// TIA Portal V18 export
TYPE "UDT_MES_Monitoring_station"
   STRUCT
      StationName : String := 'Station X';
      CheckIn : Struct
         Req : Bool;
         OK : Bool;
         NG : Bool;
         Done : Bool;
         InProgress : Bool;
         Timeout : Bool;
         Elapsed : Time;
         BothOkNg : Bool;
         UnexpectedDone : Bool;
         CountOK : UDInt;
         CountNG : UDInt;
         CountDone : UDInt;
         CountTimeout : UDInt;
         DATA : Struct
            PLC_PartTypeID : Int;
            PLC_StationRecipeNo : Int;
            PLC_StationDMXCode : String[128];
            PLC_StationStatus : Int;
            MES_ErrorCode : Int;
            MES_StatusBits : DInt;
            MES_Cycle_ID : DInt;
            MES_Unit_ParttypeID : Int;
         END_STRUCT;
      END_STRUCT;
      CheckOut : Struct
         Req : Bool;
         StoredOK : Bool;
         StoredNG : Bool;
         Done : Bool;
         InProgress : Bool;
         Timeout : Bool;
         Elapsed : Time;
         BothOkNg : Bool;
         UnexpectedDone : Bool;
         CountOK : UDInt;
         CountNG : UDInt;
         CountDone : UDInt;
         CountTimeout : UDInt;
         DATA : Struct
            PLC_PartTypeID : Int;
            PLC_StationDMXCode : String[50];
            PLC_StationRecipeNo : Int;
            PLC_PartStatus : Int;
            PLC_SubPartSN1 : String[50];
            PLC_TransferTime : String[50];
            PLC_Power : Real;
            PLC_Displacement : Real;
            PLC_Program : Int;
            PLC_NGCode : Int;
            MES_ErrorCode : Int;
            MES_ErrorMsg : String[60];
         END_STRUCT;
      END_STRUCT;
      SubPart : Struct
         OK : Bool;
         NG : Bool;
         Done : Bool;
         BothOkNg : Bool;
         CountOK : UDInt;
         CountNG : UDInt;
         CountDone : UDInt;
      END_STRUCT;
      LoadResultsStored : Struct
         OK : Bool;
         NG : Bool;
         Done : Bool;
         BothOkNg : Bool;
         CountOK : UDInt;
         CountNG : UDInt;
         CountDone : UDInt;
      END_STRUCT;
   END_STRUCT;
END_TYPE
